// TIA Portal V20 export
TYPE "UDT_EntrePLCs"
   STRUCT
      Mckey : UDInt;
      MesaDestino : UInt;   // Mesa Destino de la UT >>> RUTA[1]
      MesaSiguienteRuta : UInt;   // Mesa Siguiente >>> RUTA[0]
      Grupo : UInt;   // Numero de Grupo de la UT
      TipoCarga : USInt;   // Tipo de Carga
      AtributosDelaCarga : Struct
         Vacia : Bool;   // Atributos Especiales del la Carga --> Vacia
         Pila : Bool;   // Atributos Especiales del la Carga --> Pila
         Remontada : Bool;   // Atributos Especiales del la Carga --> Remontada
      END_STRUCT;
   END_STRUCT;
END_TYPE
